{attribute 'linkalways'} 
{attribute 'no_explicit_call' := 'This FB is a CLASS and must be accessed using methods or properties'}
{attribute 'enable_dynamic_creation'}
FUNCTION_BLOCK INTERNAL DefaultMoveBuilder IMPLEMENTS MoveBuilder
VAR
	parent_builder : MotionBuilder;
	parameters : REFERENCE TO BuilderParameters;
	move_velocity_builder : DefaultMoveVelocityBuilder(parent_builder := parent_builder, parameters := parameters);
	move_absolute_builder : DefaultMoveAbsoluteBuilder(parent_builder := parent_builder, parameters := parameters);
	move_relative_builder : DefaultMoveRelativeBuilder(parent_builder := parent_builder, parameters := parameters);
	gear_in_builder : DefaultGearInBuilder(parent_builder := parent_builder, parameters := parameters);
END_VAR

METHOD PUBLIC Acceleration : MoveBuilder
VAR_INPUT
	value : LREAL;
END_VAR
parameters.acceleration := value;
Acceleration := THIS^;
END_METHOD

METHOD PUBLIC BufferMode : MoveBuilder
VAR_INPUT
	mode : MotionBufferMode;
END_VAR
parameters.buffer_mode := mode;
BufferMode := THIS^;
END_METHOD

METHOD PUBLIC BuildHaltCommand : MotionCommand
VAR_INPUT
	axis : REFERENCE TO Mc2Axis;
END_VAR
VAR
	command_ptr : POINTER TO HaltCommand;
	command : MotionCommand;
END_VAR
command_ptr := __NEW(HaltCommand(
	axis := axis,
	deceleration := parameters.deceleration,
	jerk := parameters.jerk,
	buffer_mode := parameters.buffer_mode
));
BuildHaltCommand := command_ptr^;
END_METHOD

METHOD PUBLIC Deceleration : MoveBuilder
VAR_INPUT
	value : LREAL;
END_VAR
parameters.deceleration := value;
Deceleration := THIS^;
END_METHOD

METHOD PUBLIC Distance : MoveRelativeBuilder
VAR_INPUT
	value : LREAL;
END_VAR
parameters.distance := value;
Distance := move_relative_builder;
END_METHOD

//FB_Init is always available implicitly and it is used primarily for initialization.
//The return value is not evaluated. For a specific influence, you can also declare the
//methods explicitly and provide additional code there with the standard initialization
//code. You can evaluate the return value.
METHOD FB_Init: BOOL
VAR_INPUT
    bInitRetains : BOOL; // TRUE: the retain variables are initialized (reset warm / reset cold)
    bInCopyCode : BOOL;  // TRUE: the instance will be copied to the copy code afterward (online change)
	parent_builder : MotionBuilder;
	parameters : REFERENCE TO BuilderParameters;
END_VAR
THIS^.parent_builder := parent_builder;
THIS^.parameters REF= parameters;
END_METHOD

METHOD PUBLIC Jerk : MoveBuilder
VAR_INPUT
	value : LREAL;
END_VAR
parameters.jerk := value;
Jerk := THIS^;
END_METHOD

METHOD PUBLIC Position : MoveAbsoluteBuilder
VAR_INPUT
	value : LREAL;
END_VAR
parameters.position := value;
Position := move_absolute_builder;
END_METHOD

METHOD PUBLIC RatioDenominator : GearInBuilder
VAR_INPUT
	value : UINT;
END_VAR
parameters.ratio_denominator := value;
RatioDenominator := gear_in_builder;
END_METHOD

METHOD PUBLIC RatioNumerator : GearInBuilder
VAR_INPUT
	value : LREAL;
END_VAR
parameters.ratio_numerator := value;
RatioNumerator := gear_in_builder;
END_METHOD

METHOD PUBLIC Reset : MoveBuilder
parameters.acceleration := 0;
parameters.deceleration := 0;
parameters.jerk := 0;
parameters.buffer_mode := MotionBufferMode.Aborting;
Reset := THIS^;
END_METHOD

METHOD PUBLIC Velocity : MoveVelocityBuilder
VAR_INPUT
	value : LREAL;
END_VAR
parameters.velocity := value;
Velocity := move_velocity_builder;
END_METHOD

END_FUNCTION_BLOCK

(* stored: Version 1.1.0.1
   POU DefaultMoveBuilder: Id {7cc6e411-6752-4f2e-99f0-f4438d1a908a}, SpecialFunc None
   Folder Builders: Id {34f540d6-92b4-474e-be32-fb01f8674988}
   Folder Constructor: Id {52e2fcc3-a98f-4ee3-9141-a97ed05d40ba}
   Folder Property Setters: Id {8d89c4dc-4006-4a63-a63f-c3833a9c4fb3}
   Method Acceleration: Id {3ba4f4e3-87f3-4117-a0af-c1f0fda7c66b}
   Method BufferMode: Id {093cfb20-4e19-4b4c-a237-f1ac9b9fcb01}
   Method BuildHaltCommand: Id {b610c3c1-e30d-45a1-a3a3-8fb000d29513}
   Method Deceleration: Id {7295ce6e-e8e9-4be9-a64d-a3d271cf3adb}
   Method Distance: Id {f40db5ff-34b7-481f-9549-a30b818e4037}
   Method FB_Init: Id {6f75ec96-9124-45ed-a5a4-c413c3b30184}
   Method Jerk: Id {500c3409-5b5c-4b1c-b5c8-f6d786fa06cf}
   Method Position: Id {8a5dd1c1-c600-4226-ac69-4c19e2e8a891}
   Method RatioDenominator: Id {b3551f1c-727f-4df8-8acd-575ea808fc30}
   Method RatioNumerator: Id {50e1974e-a297-4304-b9f4-b6e58132657d}
   Method Reset: Id {d0804fb5-655e-4075-aeca-60466590d206}
   Method Velocity: Id {01ef05a0-722f-415b-adc5-4c5f4d7a6eb7} *)
